PROGRAM Oil_sort
VAR
END_VAR

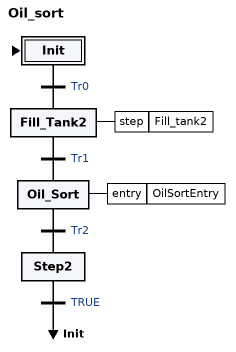
INITIAL_STEP Init:
END_STEP
TRANSITION FROM Init TO Fill_Tank2
    := Tr0;
END_TRANSITION
STEP Fill_Tank2:
    Fill_tank2(N);  // step action
END_STEP
TRANSITION FROM Fill_Tank2 TO Oil_Sort
    := Tr1;
END_TRANSITION
STEP Oil_Sort:
    OilSortEntry(P1);  // entry action
END_STEP
TRANSITION FROM Oil_Sort TO Step2
    := Tr2;
END_TRANSITION
STEP Step2:
END_STEP
TRANSITION FROM Step2 TO Init
    := TRUE;
END_TRANSITION

ACTION Fill_tank2:
main.Motor_ON_OFF := TRUE;
main.Flow_Valve_1_Percentage := 100;
main.Level_Valve_1_Percentage := 100;
main.Level_Valve_2_Percentage := 0;
main.Level_Valve_3_Percentage := 0;
END_ACTION

ACTION Oil_SortEntry:
main.Level_Valve_1_Percentage := 45;
main.StartBuffer := TRUE;
//main. START PID
END_ACTION

TRANSITION Tr0:
main.StartProcess = TRUE;
END_TRANSITION

TRANSITION Tr1:
main.LT2mm = 135;
END_TRANSITION

TRANSITION Tr2:
//main.level_3_percentage = 70;
END_TRANSITION

END_PROGRAM

(* stored: Version 1.1.0.1, ProductVersion 3.1.4024.12
   POU Oil_sort: Id {13b26af2-2d5e-4298-9f1b-77285544cb7f}, SpecialFunc None
   Action Fill_tank2: Id {4b1859af-8fdf-4c1a-8485-bf4d4700e6da}
   Action Oil_SortEntry: Id {05112cb0-9eeb-4a3d-8280-cd0bc4d72121}
   Transition Tr0: Id {dc4c5209-c520-491d-aa13-77f2dba0a3c6}
   Transition Tr1: Id {b74eb235-5d99-4277-a917-0c422f3ce085}
   Transition Tr2: Id {40f90c0d-e21f-4d5c-8422-b8ec7fddfd67} *)
